{attribute 'strict'}
{attribute 'to_string'}
TYPE E_CNC_Robot_Programs :
(
	NoCommand					:= 0, 	// Amíg "0"-ás a programszám addig nincs mozgási program végrehajtás, vár…
	Home						:= 1,	// Robot Zóna-6-ba megy és bemozog alaphelyzetbe
	Park						:= 2,	// Robot Zóna-6-ba megy és bemozog parkoló pozícióba.
	Service						:= 3,	// Robot elmegy szerviz pozícióba.
	QuickHome					:= 4,	// Robot aktuális pozícióból elmegy gyors alaphelyzetbe. (A güdelen az aktuális ponton marad a robot.)
	CNC_1_PutDown				:= 11,	// CNC 1-be rakás
	CNC_1_PickUp 				:= 12,	// CNC 1-ből kivétel
	CNC_2_PutDown 				:= 21,	// CNC 2-be rakás
	CNC_2_PickUp 				:= 22,	// CNC 2-ből kivétel
	CNC_3_PutDown 				:= 31,	// CNC 3-ba rakás
	CNC_3_PickUp  				:= 32,	// CNC 3-ból kivétel
	Lifter_1A_PickUp			:= 41,	// Kiemelő 1A-ból kiszedés
	Lifter_1A_PutDown 			:= 42,	// Kiemelő 1A-ba berakás
	Lifter_1B_PickUp			:= 43,	// Kiemelő 1B-ből kiszedés
	Lifter_1B_PutDown 			:= 44,	// Kiemelő 1B-be berakás
	Lifter_2A_PickUp			:= 51,	// Kiemelő 2A-ból kiszedés
	Lifter_2A_PutDown			:= 52,	// Kiemelő 2A-ba berakás
	Lifter_2B_PickUp			:= 53,	// Kiemelő 2B-ből kiszedés
	Lifter_2B_PutDown  			:= 54,	// Kiemelő 2B-be berakás
	Lifter_3A_PickUp			:= 61,	// Kiemelő 3A-ból kiszedés
	Lifter_3A_PutDown  			:= 62,	// Kiemelő 3A-ba berakás
	Lifter_3B_PickUp 			:= 63,	// Kiemelő 3B-ből kiszedés
	Lifter_3B_PutDown 			:= 64,	// Kiemelő 3B-be berakás
	Lifter_1A_Camera			:= 71,	// Kiemelő 1A-nál kamerázás
	Lifter_1B_Camera 			:= 72,	// Kiemelő 1B-nél kamerázás
	Lifter_2A_Camera			:= 73,	// Kiemelő 2A-nál kamerázás
	Lifter_2B_Camera			:= 74,	// Kiemelő 2B-nél kamerázás
	Lifter_3A_Camera			:= 75,	// Kiemelő 3A-nál kamerázás
	Lifter_3B_Camera 			:= 76,	// Kiemelő 3B-nél kamerázás
	Master_Part_PickUp			:= 101,
	Master_Part_PutDown			:= 102,
	Lifter_1A_Master_PickUp		:= 111,
	Lifter_1A_Master_PutDown	:= 112,
	Lifter_1B_Master_PickUp		:= 113,
	Lifter_1B_Master_PutDown	:= 114,
	Lifter_2A_Master_PickUp 	:= 121,
	Lifter_2A_Master_PutDown	:= 122,
	Lifter_2B_Master_PickUp 	:= 123,
	Lifter_2B_Master_PutDown	:= 124,
	Lifter_3A_Master_PickUp		:= 131,
	Lifter_3A_Master_PutDown	:= 132,
	Lifter_3B_Master_PickUp		:= 133,
	Lifter_3B_Master_PutDown 	:= 134
);
END_TYPE

(* stored: Version 1.1.0.1, ProductVersion 3.1.4024.12
   EnumerationTextList E_CNC_Robot_Programs: Id {91f25d92-4e02-47d4-ae40-64b374991344} *)
